{attribute 'qualified_only'}
VAR_GLOBAL CONSTANT
    PortNo : UINT := 852;
END_VAR

(* stored: Version 1.1.0.1, ProductVersion 3.1.4024.9
   GVL Constants: Id {320a0642-6429-0b7c-27af-b9f64592c9af} *)
